(*udt (user defined type) for all KUKA KRC4 Robot systems on EL6692 ECAT Bridge
	Author(S): Brent Lekx-Toniolo of Sodecia GTAC;
	Version 1.0: November 2012
		- Initial Concept
	Version 20121204
		Changes from v1
			- Change to Naming Convention to include date as version

	Last Edit: December 4th, 2012, blt
*)
TYPE udt_EtherCAT_Kuka_OutputBits_20121204 :
STRUCT
	Robot_IN: ARRAY [1..512] OF BOOL;
END_STRUCT
END_TYPE

(* stored: Version 1.1.0.1, ProductVersion 3.1.4024.5
   DUT udt_EtherCAT_Kuka_OutputBits_20121204: Id {06d7ee4b-804f-466b-b49d-e5886e82fd13} *)
